(* IEC 61131-3 sources: F100R_S278_Temperville/MyController.device.xml.v3^/Plc Logic.plclogic.xml.v3^/Application.application.xml.v3^/03_Geral, 12 files *)

(* ---- B_Imagens.prg.st ---- *)
PROGRAM B_Imagens
VAR
	Index: INT;
END_VAR

//Imagens de Motores
ImgMotor[1]:=xMotorEntradaLigado;
ImgMotor[2]:=ImgMotor[2];
ImgMotor[3]:=xMotorFornoLigado;
ImgMotor[4]:=xMotorPassagemLigado;
ImgMotor[5]:=xMotorResfriadorLigado;
ImgMotor[6]:=xMotorSaidaLigado;
ImgMotor[7]:=xMotorDifusorSup01Ligado;
ImgMotor[8]:=xMotorDifusorInf01Ligado;
ImgMotor[9]:=xMotorDifusorSup02Ligado;
ImgMotor[10]:=xMotorDifusorInf02Ligado;
ImgMotor[11]:=xMotorGuilhotina01Ligado;
ImgMotor[12]:=xMotorGuilhotina02Ligado;
ImgMotor[13]:=xMotorLimpResfr02Ligado;
ImgMotor[14]:=xMotorCaixaFornoLigado;
ImgMotor[15]:=xMotorVentilador01Ligado;
ImgMotor[16]:=xMotorVentilador02Ligado;
ImgMotor[17]:=xMotorVentilador03Ligado;
ImgMotor[18]:=xMotorVentilador04Ligado;
ImgMotor[19]:=xMotorVentilador04Ligado;
ImgMotor[20]:=xMotorVentConvecEntLigado;
ImgMotor[21]:=xMotorVentConvecSaiLigado;
ImgMotor[22]:=xMotorGuilhotina01SupLigado;
ImgMotor[23]:=xMotorGuilhotina01InfLigado;
ImgMotor[24]:=xKaMotorOscilaResfr02Sup;
ImgMotor[25]:=xKaMotorOscilaResfr02Inf;

//Imagens de Válvula
ImgValvAberta[1]:=xSensorPortaEntrada;
ImgValvAberta[2]:=xSensorPortaSaida;
ImgValvAberta[3]:=xValvulaConveccaoLigada;
ImgValvAberta[4]:=xSensorGradeEntradaUp;
ImgValvAberta[5]:=xSensorGradeSaidaUp;

ImgValvFechada[1]:= NOT xSensorPortaEntrada;
ImgValvFechada[2]:= NOT xSensorPortaSaida;
ImgValvFechada[3]:= NOT xValvulaConveccaoLigada;
ImgValvFechada[4]:=	NOT xSensorGradeEntradaUp;
ImgValvFechada[5]:=	NOT xSensorGradeSaidaUp;

//Imagens Gerais
ImgGeral[1]:=xStatusNobreak;
ImgGeral[2]:=xBt01Emergencia; // Mesa Computador
ImgGeral[3]:=xBt02Emergencia; // Mesa Manual
ImgGeral[4]:=xBt03Emergencia; //
ImgGeral[5]:=xBt04Emergencia;
ImgGeral[6]:=xBt05Emergencia;
ImgGeral[7]:=xBt06Emergencia;
ImgGeral[8]:=xBt07Emergencia;
ImgGeral[9]:=xBt08Emergencia;
ImgGeral[10]:=xBt09Emergencia;
ImgGeral[11]:=xBt10Emergencia;
ImgGeral[12]:=xVentiladoresPainel;
ImgGeral[13]:=xVentiladoresSsr;
ImgGeral[14]:=xValvulaVeneziana;

FOR Index:=1 TO iNumResistencias DO
//	ImgRetornoSsrInferior[Index]:=xRetornoSsrInferior[Index];
//	ImgRetornoSsrSuperior[Index]:=xRetornoSsrSuperior[Index];
//	ImgResistenciaInferior[Index]:=xResistenciaInferior[Index];
//	ImgResistenciaSuperior[Index]:=xResistenciaSuperior[Index];
	ImgRetornoSsrInferior[Index]:=xResistenciaInferior[Index];
	ImgRetornoSsrSuperior[Index]:=xResistenciaSuperior[Index];
	ImgResistenciaHabilitadaInferior[Index]:=xResistenciaHabilitadaInferior[Index];
	ImgResistenciaHabilitadaSuperior[Index]:=xResistenciaHabilitadaSuperior[Index];
END_FOR

(* ---- C_Alarmes.prg.st ---- *)
PROGRAM C_Alarmes
VAR
	IndexAlm01: INT;
	AlmValvPortaEntrada: AlarmeValvula1vNeg;
	AlmValvPortaSaida: AlarmeValvula1vNeg;
	AlmGradeEntrada: AlarmeValvula1v;
	AlmGradeSaida: AlarmeValvula1v;
	TpAlmMotorSom: ARRAY[1..25] OF TP;
	TpAlmMotorSomIn: ARRAY[1..25] OF BOOL;
	TpAlmMotorSomQ: ARRAY[1..25] OF BOOL;
	AlmMotorSom: ARRAY[1..25] OF BOOL;
	AlarmeSom: TimerGeneration;
	AlarmeLum: TimerGeneration;
	xAlarmeSomEnable: BOOL;
	xAlarmeSomOut: BOOL;
	xAlarmeLumEnable: BOOL;
	xAlarmeLumOut: BOOL;
	TpRstSuper: TP;
	TpRstSuperiN: BOOL;
	TpRstSuperQ: BOOL;
	xAlarmeSonPortaEntradaForno: BOOL;
	xAlarmeSonPortaSaidaForno: BOOL;
	xAlarmeSonValvulaGradeEntrada: BOOL;
	xAlarmeSonValvulaGradeSaida: BOOL;
	xAlarmeGeralEncoder: BOOL;
	xAlarmeSonoroEncoderGeral: BOOL;
	xAlarmeGeralMotorParado: BOOL;
	xAlarmeSonoroMotorParadoGeral: BOOL;
	AlmMotoresBitsSoma: INT;
	AlmMotoresSonBitsSoma: INT;
END_VAR

AlmMotoresBitsSoma:=0;
AlmMotoresSonBitsSoma:=0;
FOR IndexAlm01:=1 TO 50 DO
	xAlarmesResistenciasGeralInferior[IndexAlm01]:=xAlarmeSsrInferiorFechado[IndexAlm01] OR xAlarmeSsrInferiorAberto[IndexAlm01] OR (*xAlarmeResistRompidaInferior[IndexAlm01]*) xFalhaForcadaInferior[IndexAlm01] OR xAlarmeResistForceInferior[IndexAlm01] OR AlmTermoparAbertoLogicoInf[IndexAlm01] OR AlmTemperaturaExcedeuLogicoInf[IndexAlm01];
	xAlarmesResistenciasGeralSuperior[IndexAlm01]:=xAlarmeSsrSuperiorFechado[IndexAlm01] OR xAlarmeSsrSuperiorAberto[IndexAlm01] OR (*xAlarmeResistRompidaSuperior[IndexAlm01]*) xFalhaForcadaSuperior[IndexAlm01] OR xAlarmeResistForceSuperior[IndexAlm01] OR AlmTermoparAbertoLogicoSup[IndexAlm01] OR AlmTemperaturaExcedeuLogicoSup[IndexAlm01];

	AlmMotoresBitsSoma:= AlmMotoresBitsSoma+ BOOL_TO_INT (AlmMotor[IndexAlm01]);

	TpAlmMotorSomIn[IndexAlm01]:=AlmMotor[IndexAlm01];
	TpAlmMotorSom[IndexAlm01](IN:=TpAlmMotorSomIn[IndexAlm01] , PT:=T#1S , Q=>TpAlmMotorSomQ[IndexAlm01] , ET=> );
	IF TpAlmMotorSomQ[IndexAlm01] THEN
		AlmMotorSom[IndexAlm01]:=TRUE;
	END_IF
	IF	bResetAlmGeral or xResetErro THEN
		AlmMotorSom[IndexAlm01]:=FALSE;
		AlmMotoresSonBitsSoma:=0;

	END_IF
	AlmMotoresSonBitsSoma:= AlmMotoresSonBitsSoma+ BOOL_TO_INT (AlmMotorSom[IndexAlm01]);

	xAlarmesTestesResistenciasInferiores[IndexAlm01]:=xTesteResistenciaInferiorFlh[IndexAlm01] OR xFalhaForcadaInferior[IndexAlm01] OR xAlarmeResistForceInferior[IndexAlm01];
	xAlarmesTestesResistenciasSuperiores[IndexAlm01]:=xTesteResistenciaSuperiorFlh[IndexAlm01] OR xFalhaForcadaSuperior[IndexAlm01] OR xAlarmeResistForceSuperior[IndexAlm01];

END_FOR;
xAlarmesMotores:= AlmMotoresBitsSoma>=1;
xAlarmesMotoresSon:= AlmMotoresSonBitsSoma>=1;

TpRstSuper(IN:=BtResetAlarmesGerais , PT:=T#500MS , Q=> TpRstSuperQ, ET=> );

bResetAlmGeral:=TpRstSuperQ OR xBtCalaAlarme ;
xBotaoResetaDrives:=TpRstSuperQ OR xBtCalaAlarme ;

IF BtResetAlarmesGerais THEN
	BtResetAlarmesGerais:=FALSE;
END_IF
//Alarmes de Motores

xAlarmeMotorEntrada	:=(xFalhaMotorEntrada OR xAlarmeCofInverMesaEntra);//AND NOT xPausaEmergenciaTof;
xAlarmeMotorForno	:=(xFalhaMotorForno OR xAlarmeCofInverMesaForno);//AND NOT xPausaEmergenciaTof;
xAlarmeMotorPass	:=(xFalhaMotorPassagem );//AND NOT xPausaEmergenciaTof;
xAlarmeMotorResfriador:=(xFalhaMotorResfriador OR xAlarmeCofInverMesaResfr);//AND NOT xPausaEmergenciaTof;
xAlarmeMotorSaida	:=(xFalhaMotorSaida OR xAlarmeCofInverMesaSaida);//AND NOT xPausaEmergenciaTof;
xAlarmeMotorDifusorInf01:=(xFalhaMotorDifusorInf01 );//AND NOT xPausaEmergenciaTof;
xAlarmeMotorDifusorSup01:=(xFalhaMotorDifusorSup01 );//AND NOT xPausaEmergenciaTof;
xAlarmeMotorDifusorInf02:=(xFalhaMotorDifusorInf02 );//AND NOT xPausaEmergenciaTof;
xAlarmeMotorDifusorSup02:=(xFalhaMotorDifusorSup02 OR xAlarmeCofInverResfrSup02);//AND NOT xPausaEmergenciaTof;
xAlarmeMotorGuilhotina01:=(xFalhaMotorGuilhotina01 );//AND NOT xPausaEmergenciaTof;
xAlarmeMotorGuilhotina02:=(xFalhaMotorGuilhotina02 OR xAlarmeCofInverGuilho02);//AND NOT xPausaEmergenciaTof;
xAlarmeMotorLimpResfr02:=(xFalhaMotorLimpResfr02 );//AND NOT xPausaEmergenciaTof;
xAlarmeMotorCaixaForno:=(xFalhaMotorCaixaForno OR xAlarmeCofInverCaixaForno);//AND NOT xPausaEmergenciaTof;
xAlarmeMotorVentilador01:=(xFalhaMotorVentilador01 );//AND NOT xPausaEmergenciaTof;
xAlarmeMotorVentilador02:=(xFalhaMotorVentilador02 );//AND NOT xPausaEmergenciaTof;
xAlarmeMotorVentilador03:=(xFalhaMotorVentilador03 OR xAlarmeCofInverVentila03);//AND NOT xPausaEmergenciaTof;
xAlarmeMotorVentilador04:=(xFalhaMotorVentilador04 );//AND NOT xPausaEmergenciaTof;
xAlarmeMotorVentConvecEnt:=(xFalhaMotorVentConvecEnt OR xAlarmeCofInverConvecEnt);//AND NOT xPausaEmergenciaTof;
xAlarmeMotorVentConvecSai:=(xFalhaMotorVentConvecSai );//AND NOT xPausaEmergenciaTof;
xAlarmeMotorGuilhotina01Sup:=(xFalhaMotorGuilhotina01Sup );//AND NOT xPausaEmergenciaTof;
xAlarmeMotorGuilhotina01Inf:=(xFalhaMotorGuilhotina01Inf );//AND NOT xPausaEmergenciaTof;

AlmMotor[1]:=xAlarmeMotorEntrada;
AlmMotor[2]:=AlmMotor[2];
AlmMotor[3]:=xAlarmeMotorForno;
AlmMotor[4]:=xAlarmeMotorPass;
AlmMotor[5]:=xAlarmeMotorResfriador;
AlmMotor[6]:=xAlarmeMotorSaida;
AlmMotor[7]:=xAlarmeMotorDifusorSup01;
AlmMotor[8]:=xAlarmeMotorDifusorInf01;
AlmMotor[9]:=xAlarmeMotorDifusorSup02;
AlmMotor[10]:=xAlarmeMotorDifusorInf02;
AlmMotor[11]:=xAlarmeMotorGuilhotina01;
AlmMotor[12]:=xAlarmeMotorGuilhotina02;
AlmMotor[13]:=AlmMotor[13];
AlmMotor[14]:=xAlarmeMotorCaixaForno;
AlmMotor[15]:=xAlarmeMotorVentilador01;
AlmMotor[16]:=xAlarmeMotorVentilador02;
AlmMotor[17]:=xAlarmeMotorVentilador03;
AlmMotor[18]:=xAlarmeMotorVentilador04;
AlmMotor[19]:=xAlarmeMotorBombaHidraulica;
AlmMotor[20]:=xAlarmeMotorVentConvecEnt;
AlmMotor[21]:=xAlarmeMotorVentConvecSai;
AlmMotor[22]:=xAlarmeMotorGuilhotina01Sup;
AlmMotor[23]:=xAlarmeMotorGuilhotina01Inf;
AlmMotor[24]:=xAlarmeMotorOscilaSup02;
AlmMotor[25]:=xAlarmeMotorOscilaInf02;

//Alarmes de Válvula

xSensorPortaEntradaAberta:=xSensorPortaEntrada;
xSensorPortaEntradaFechada:= NOT xSensorPortaEntrada;

AlmValvPortaEntrada(
	SensorValvAberta:= xSensorPortaEntradaAberta ,
	SensorValvFechad:= xSensorPortaEntradaFechada,
	AcionamentoValvula:= xValvPortaEntradaForno,// OR xOperacaoManual,
	ResetAlarm:=bResetAlmGeral OR xOperacaoManual,
	TempoAberto:= T#1500MS,
	TempoFechad:= T#1500MS,
	AlarmeValvAberta=> xAlarmePortaEntradaFornoAberta, //Porta não Abriu
	AlarmeValvFechada=> xAlarmePortaEntradaFornoFechada, // Porta não Fechou
	AlarmeSonoro=> xAlarmeSonPortaEntradaForno);

xAlarmePortaEntradaForno:=xAlarmePortaEntradaFornoAberta OR xAlarmePortaEntradaFornoFechada;

xSensorPortaSaidaAberta:=xSensorPortaSaida;
xSensorPortaSaidaFechada:= NOT xSensorPortaSaida;

AlmValvPortaSaida(
	SensorValvAberta:= xSensorPortaSaidaAberta ,
	SensorValvFechad:= xSensorPortaSaidaFechada,
	AcionamentoValvula:= xValvPortaSaidaForno,// OR xOperacaoManual,
	ResetAlarm:=bResetAlmGeral OR xOperacaoManual,
	TempoAberto:= T#2500MS,
	TempoFechad:= T#2000MS,
	AlarmeValvAberta=> xAlarmePortaSaidaFornoAberta, //Porta não Abriu
	AlarmeValvFechada=> xAlarmePortaSaidaFornoFechada, // Porta não Fechou
	AlarmeSonoro=> xAlarmeSonPortaSaidaForno);

xAlarmePortaSaidaForno:=xAlarmePortaSaidaFornoAberta OR xAlarmePortaSaidaFornoFechada;

// Alarme Grade Mesa de Entrada

xSensorGradeEntradaDown:= NOT xSensorGradeEntradaUp;

(*
AlmGradeEntrada(
	SensorValvAberta:= xSensorGradeEntradaUp,
	SensorValvFechad:= xSensorGradeEntradaDown,
	AcionamentoValvula:= xValvulaGradeEntrada,
	ResetAlarm:=bResetAlmGeral,
	TempoAberto:= T#2000MS,
	TempoFechad:= T#2000MS,
	AlarmeValvAberta=> xAlarmeValvulaGradeEntradaUp,
	AlarmeValvFechada=> xAlarmeValvulaGradeEntradaDown,
	AlarmeSonoro=>xAlarmeSonValvulaGradeEntrada);
*)
xAlarmeValvulaGradeEntrada:= xAlarmeValvulaGradeEntradaUp OR xAlarmeValvulaGradeEntradaDown;

// Alarme Grade Mesa de Saída

xSensorGradeSaidaDown:= NOT xSensorGradeSaidaUp;

AlmGradeSaida(
	SensorValvAberta:= xSensorGradeSaidaUp,
	SensorValvFechad:= xSensorGradeSaidaDown,
	AcionamentoValvula:= xValvulaGradeSaida,
	ResetAlarm:=bResetAlmGeral,
	TempoAberto:= T#5000MS,
	TempoFechad:= T#4000MS,
	AlarmeValvAberta=> xAlarmeValvulaGradeSaidaUp,
	AlarmeValvFechada=> xAlarmeValvulaGradeSaidaDown,
	AlarmeSonoro=> xAlarmeSonValvulaGradeSaida);

xAlarmeValvulaGradeSaida:= xAlarmeValvulaGradeSaidaUp OR xAlarmeValvulaGradeSaidaDown;

AlmValvAberta[1]:=xAlarmePortaEntradaFornoAberta;
AlmValvAberta[2]:=xAlarmePortaSaidaFornoAberta;
AlmValvAberta[3]:=xAlarmeValvulaGradeEntradaUp;
AlmValvAberta[4]:=xAlarmeValvulaGradeSaidaUp;
AlmValvAberta[5]:=AlmValvAberta[5];
AlmValvAberta[6]:=AlmValvAberta[6];
AlmValvAberta[7]:=AlmValvAberta[7];
AlmValvAberta[8]:=AlmValvAberta[8];
AlmValvAberta[9]:=AlmValvAberta[9];
AlmValvAberta[10]:=AlmValvAberta[10];

AlmValvFechada[1]:=xAlarmePortaEntradaFornoFechada;
AlmValvFechada[2]:=xAlarmePortaSaidaFornoFechada;
AlmValvFechada[3]:=xAlarmeValvulaGradeEntradaDown;
AlmValvFechada[4]:=xAlarmeValvulaGradeSaidaDown;
AlmValvFechada[5]:=AlmValvFechada[5];
AlmValvFechada[6]:=AlmValvFechada[6];
AlmValvFechada[7]:=AlmValvFechada[7];
AlmValvFechada[8]:=AlmValvFechada[8];
AlmValvFechada[9]:=AlmValvFechada[9];
AlmValvFechada[10]:=AlmValvFechada[10];

//Alarmes Gerais
AlmGeral[1]:=xAlarmePressaoArBaixaRede;
AlmGeral[2]:=xAlarmePressaoArAltaRede;
AlmGeral[3]:=xAlmNobreak;
AlmGeral[4]:=xSemEnergia;
AlmGeral[5]:=xLimpVidroForaPosicao;
AlmGeral[6]:=xAlmDisjGeral;
AlmGeral[7]:=xAlmDisjResist;
AlmGeral[8]:=xAlarmePressaoArBaixaMaq;
AlmGeral[9]:=xAlarmePressaoArAltaMaq;
AlmGeral[10]:=AlmGeral[10];

// Alarmes de Encoder
xAlarmeGeralEncoder:= xAlarmeGeralEncoderMeForno OR xAlarmeGeralEncoderMeResfriador (*OR xAlarmeGeralEncoderDuResfriadorSup01 OR xAlarmeGeralEncoderDuResfriadorInf01*) OR xAlarmeGeralEncoderDuResfriadorSup02 (*OR xAlarmeGeralEncoderDuResfriadorInf02 OR xAlarmeGeralEncoderGuiResfriador01*) OR xAlarmeGeralEncoderGuiResfriador02;
xAlarmeSonoroEncoderGeral:= xAlarmeSonoroEncoderMeForno OR xAlarmeSonoroEncoderMeResfriador (*OR xAlarmeSonoroEncoderDuResfriadorSup01 OR xAlarmeSonoroEncoderDuResfriadorInf01*) OR xAlarmeSonoroEncoderDuResfriadorSup02 (*OR xAlarmeSonoroEncoderDuResfriadorInf02 OR xAlarmeSonoroEncoderGuiResfriador01*) OR xAlarmeSonoroEncoderGuiResfriador02;

AlmEncoder[1]:=AlmEncoder[1];
AlmEncoder[2]:=xAlarmeGeralEncoderMeForno;
AlmEncoder[3]:=xAlarmeGeralEncoderMeResfriador;
AlmEncoder[4]:=xAlarmeGeralEncoderDuResfriadorSup01;
AlmEncoder[5]:=FALSE;//xAlarmeGeralEncoderDuResfriadorInf01;
AlmEncoder[6]:=xAlarmeGeralEncoderDuResfriadorSup02;
AlmEncoder[7]:=xAlarmeGeralEncoderDuResfriadorInf02;
AlmEncoder[8]:=xAlarmeGeralEncoderGuiResfriador01;
AlmEncoder[9]:=xAlarmeGeralEncoderGuiResfriador02;
AlmEncoder[10]:=FALSE;

// Alarmes Motor Parado por Falha Desconhecida

xAlarmeGeralMotorParado:=  xAlarmeMeFornoParado OR xAlarmeMeResfrParado;
xAlarmeSonoroMotorParadoGeral:= xAlarmeMeFornoParadoSom OR xAlarmeMeResfrParadoSom;

AlmMotorParado[1]:=AlmMotorParado[1];
AlmMotorParado[2]:=xAlarmeMeFornoParado;
AlmMotorParado[3]:=xAlarmeMeResfrParado;
AlmMotorParado[4]:=AlmMotorParado[4];
AlmMotorParado[5]:=AlmMotorParado[5];
AlmMotorParado[6]:=AlmMotorParado[6];
AlmMotorParado[7]:=AlmMotorParado[7];
AlmMotorParado[8]:=AlmMotorParado[8];
AlmMotorParado[9]:=AlmMotorParado[9];
AlmMotorParado[10]:=AlmMotorParado[10];

//Alerta Luminoso e Sonoro de Alarme

xAlarmeLumEnable:=xAlarmePortaEntradaForno OR xAlarmePortaSaidaForno OR xAlarmeValvulaGradeEntrada OR xAlarmeValvulaGradeSaida OR xAlarmesTermopares OR xAlarmesSSr OR xAlarmesMotores OR xAlarmePressaoArRede OR xAlarmePressaoArMaq OR xAlmNobreak OR xSemEnergia OR xAlmDisjGeral OR xAlmDisjResist OR xAlarmeGeralEncoder OR xAlarmeGeralMotorParado OR xLimpVidroForaPosicao OR xAlarmeSsrConvecEntSin OR xAlmTermoparAbertoConvecEntSin OR xAlmTemperExcedeuConvecEntSin;
AlarmeLum(ENABLE:=xAlarmeLumEnable , TIMELOW:=T#1S , TIMEHIGH:=T#1S , OUT=>xAlarmeLumOut );
//xAlarmeLuminoso:=xAlarmeLumOut OR xBtEmergencia OR NOT xReleSeguranca;
xSinalLumAmar:=xAlarmeLumOut;
xSinalLumVerm:=xBtEmergencia OR NOT xReleSeguranca OR xLedMotFornoStop;
xSinalLumVerd:= NOT xSinalLumVerm AND xLedMaqEmCiclo;

xAlarmeSomEnable:=xAlarmeSonPortaEntradaForno OR xAlarmeSonPortaSaidaForno OR xAlarmeSonValvulaGradeSaida OR xAlarmeSonValvulaGradeEntrada OR xAlarmesTermoparesSon OR xAlarmesSSrSon OR xAlarmesMotoresSon OR xAlarmePressaoArRedeSom OR xAlarmePressaoArMaqSom OR xAlmNobreakSom OR xAlmSomSemEnergia OR xAlmDisjGeralSom OR xAlmDisjResistSom OR xAlarmeSonoroEncoderGeral OR xAlarmeSonoroMotorParadoGeral OR xLimpVidroForaPosicaoSon OR xAlarmeSsrConvecEntSon OR xAlmTermoparAbertoConvecEntSon OR xAlmTemperExcedeuConvecEntSon;
AlarmeSom(ENABLE:=xAlarmeSomEnable , TIMELOW:=T#1S , TIMEHIGH:=T#1S , OUT=>xAlarmeSomOut );

xAlarmeSonoro:= (xAlarmeSomOut OR xSomDescarga OR xSomSemEnergia AND NOT xMotorCaixaFornoLigado) OR xAlertaSomCxForno;

(* ---- D_AnimaGeralResistencias.prg.st ---- *)
PROGRAM D_AnimaGeralResistencias
VAR
	Index: INT;
END_VAR

FOR Index:=1 TO iNumResistencias DO

//xAlarmesResistenciasGeral[Index]:=xAlarmeSsrInferiorFechado[Index] OR xAlarmeSsrInferiorAberto[Index] OR xAlarmeResistRompidaInferior[Index] OR AlmTermoparAbertoLogicoInf[Index] OR AlmTemperaturaExcedeuLogicoInf[Index];
//Inferior
	IF NOT xResistenciaHabilitadaInferior[Index] AND NOT xAlarmesResistenciasGeralInferior[Index] THEN
			iAnimaResistenciaInferior[Index]:=0;(*Resistência Desabilitada*)
	END_IF
	IF NOT xResistenciaInferior[Index] AND xResistenciaHabilitadaInferior[Index]THEN
			iAnimaResistenciaInferior[Index]:=1;(*Resistência Desligada*)
	END_IF
	IF xResistenciaInferior[Index] AND xResistenciaHabilitadaInferior[Index]THEN
			iAnimaResistenciaInferior[Index]:=2; (*Resistência Ligada*)
	END_IF
	IF xFalhaForcadaInferior[Index] OR  xAlarmesResistenciasGeralInferior[Index] (*xAlarmeResistForceSuperior[Index]*) THEN
			iAnimaResistenciaInferior[Index]:=3; (*Resistência Alarme*)
	END_IF

	IF AlmTermoparAbertoLogicoInf[Index] OR AlmTemperaturaExcedeuLogicoInf[Index] THEN
			iAnimaResistenciaInferior[Index]:=4; (*Termopar Alarme*)
	END_IF

	IF xResistenciaForcadaInferior[Index] AND ValorAmperagemResistenciaInferior[Index]>5 (*xResistenciaInferior[Index]*)  (*AND xResistenciaHabilitadaInferior[Index]*) THEN
			iAnimaResistenciaInferior[Index]:=5; (*Resistência Forçada*)
	END_IF

//Superior
	IF NOT xResistenciaHabilitadaSuperior[Index] AND NOT xAlarmesResistenciasGeralSuperior[Index] THEN
			iAnimaResistenciaSuperior[Index]:=0;(*Resistência Desabilitada*)
	END_IF
	IF NOT xResistenciaSuperior[Index] AND xResistenciaHabilitadaSuperior[Index]THEN
			iAnimaResistenciaSuperior[Index]:=1;(*Resistência Desligada*)
	END_IF
	IF (*(xReleSsrSuperior[Index] OR xSaidaReleRampaPatamarSup[Index])*)xResistenciaSuperior[Index] AND xResistenciaHabilitadaSuperior[Index]THEN
			iAnimaResistenciaSuperior[Index]:=2; (*Resistência Ligada*)
	END_IF
	IF xFalhaForcadaSuperior[Index] OR (*xAlarmeResistForceSuperior[Index]*) xAlarmesResistenciasGeralSuperior[Index] THEN
			iAnimaResistenciaSuperior[Index]:=3; (*Resistência Alarme*)
	END_IF
	IF AlmTermoparAbertoLogicoSup[Index] OR AlmTemperaturaExcedeuLogicoSup[Index] THEN
			iAnimaResistenciaSuperior[Index]:=4; (*Termopar Alarme*)
	END_IF
	IF xResistenciaForcadaSuperior[Index] AND ValorAmperagemResistenciaSuperior[Index]>5 (*xResistenciaSuperior[Index]*) (*AND xResistenciaHabilitadaSuperior[Index]*) THEN
			iAnimaResistenciaSuperior[Index]:=5; (*Resistência Forçada*)
	END_IF

END_FOR

(* ---- E_AnimaTesteGeralResistencias.prg.st ---- *)
PROGRAM E_AnimaTesteGeralResistencias
VAR
	Index: INT;
END_VAR

FOR Index:=1 TO iNumResistencias DO
//Inferior
	IF NOT xAlarmesResistenciasGeralInferior[Index] AND NOT xTesteResistenciaInferiorFlh[Index] AND NOT  xResistenciaInferior[Index] AND NOT xTestandoResistenciaInferior[Index]THEN
		iAnimaTesteResistenciaInferior[Index]:=0;(*Resistência Desligada*)
	END_IF

	IF xResistenciaForcadaInferior[Index] AND ValorAmperagemResistenciaInferior[Index]>40(*xResistenciaInferior[Index]*) THEN
		iAnimaTesteResistenciaInferior[Index]:=1; (*Resistência Forçada*)
	END_IF

	IF xResistenciaInferior[Index] AND xTestandoResistenciaInferior[Index]THEN
		iAnimaTesteResistenciaInferior[Index]:=2; (*Resistência Testando*)
	END_IF

	IF xTesteResistenciaInferiorOk[Index]THEN
		iAnimaTesteResistenciaInferior[Index]:=3; (* Teste Resistência Ok*)
	END_IF

	IF xFalhaForcadaInferior[Index] OR (*xAlarmeResistForceInferior[Index]*) xAlarmesResistenciasGeralInferior[Index] OR xTesteResistenciaInferiorFlh[Index] THEN
		iAnimaTesteResistenciaInferior[Index]:=4; (* Teste Resistência Resistência Alarme*)
	END_IF

//Superior
	IF NOT xAlarmesResistenciasGeralSuperior[Index] AND NOT xTesteResistenciaSuperiorFlh[Index] AND NOT xResistenciaSuperior[Index] AND NOT xTestandoResistenciaSuperior[Index]THEN
		iAnimaTesteResistenciaSuperior[Index]:=0;(*Resistência Desligada*)
	END_IF

	IF xResistenciaForcadaSuperior[Index] AND ValorAmperagemResistenciaSuperior[Index]>40(*xResistenciaSuperior[Index]*) THEN
		iAnimaTesteResistenciaSuperior[Index]:=1; (*Resistência Forçada*)
	END_IF

	IF xResistenciaSuperior[Index] AND xTestandoResistenciaSuperior[Index]THEN
		iAnimaTesteResistenciaSuperior[Index]:=2; (*Resistência Testando*)
	END_IF

	IF xTesteResistenciaSuperiorOk[Index]THEN
		iAnimaTesteResistenciaSuperior[Index]:=3; (* Teste Resistência Ok*)
	END_IF

	IF xFalhaForcadaSuperior[Index] OR (*xAlarmeResistForceSuperior[Index]*) xAlarmesResistenciasGeralSuperior[Index] OR xTesteResistenciaSuperiorFlh[Index] THEN
		iAnimaTesteResistenciaSuperior[Index]:=4; (* Teste Resistência Resistência Alarme*)
	END_IF

END_FOR

(* ---- F_AnimaAlmMotValv.prg.st ---- *)
PROGRAM F_AnimaAlmMotValv
VAR
	Index: INT;
END_VAR

FOR Index:=1 TO 25 DO
//Motores
	IF NOT AlmMotor[Index] AND NOT ImgMotor[Index] THEN
		iAnimaAlarmesMotores[Index]:=0; //Desligado
	END_IF
	IF NOT AlmMotor[Index] AND ImgMotor[Index] THEN
		iAnimaAlarmesMotores[Index]:=1; //Ligado
	END_IF
	IF AlmMotor[Index] THEN
		iAnimaAlarmesMotores[Index]:=2; //Alarme
	END_IF
//Válvulas

	IF (NOT AlmValvAberta[Index] OR NOT AlmValvFechada[Index] ) AND ImgValvFechada[Index] THEN
		iAnimaAlarmesValvulas[Index]:=0; // Fechada
	END_IF
	IF (NOT AlmValvAberta[Index] OR NOT AlmValvFechada[Index] ) AND ImgValvAberta[Index] THEN
		iAnimaAlarmesValvulas[Index]:=1; // Aberta
	END_IF
	IF AlmValvAberta[Index] OR AlmValvFechada[Index]  THEN
		iAnimaAlarmesValvulas[Index]:=2; // Alarme
	END_IF
END_FOR

(* ---- F_MensagemErroMotor.prg.st ---- *)
PROGRAM F_MensagemErroMotor
VAR
	Index: INT;
	sCodigoErroMotor: ARRAY[1..25] OF STRING;
	sDescricaoErroMotor: ARRAY[1..25] OF STRING;
END_VAR

FOR Index:=1 TO 20 DO
	IF wErroMotorId[Index]=4096 THEN
		sCodigoErroMotor[Index]:='OLF';
		sDescricaoErroMotor[Index]:='Sobrecarga Motor ';
	END_IF
	IF wErroMotorId[Index]=8976 THEN
		sCodigoErroMotor[Index]:='OCF';
		sDescricaoErroMotor[Index]:='Sobrecorrente Motor ';
	END_IF
	IF wErroMotorId[Index]=8992 THEN
		sCodigoErroMotor[Index]:='SCF';
		sDescricaoErroMotor[Index]:='Curto Circuito Motor ';
	END_IF
	IF wErroMotorId[Index]=9008 THEN
		sCodigoErroMotor[Index]:='SCF';
		sDescricaoErroMotor[Index]:='Curto Circuito Motor (Fase-Terra) ';
	END_IF
	IF wErroMotorId[Index]=9024 THEN
		sCodigoErroMotor[Index]:='SCF';
		sDescricaoErroMotor[Index]:='Curto Circuito Motor (Fase-Fase) ';
	END_IF
	IF wErroMotorId[Index]=12560 THEN
		sCodigoErroMotor[Index]:='OSF';
		sDescricaoErroMotor[Index]:='Sobretensão na Alimentação do Motor ';
	END_IF
	IF wErroMotorId[Index]=12576 THEN
		sCodigoErroMotor[Index]:='USF';
		sDescricaoErroMotor[Index]:='Sobretensão na Alimentação do Motor ';
	END_IF
	IF wErroMotorId[Index]=12592 THEN
		sCodigoErroMotor[Index]:='PHF';
		sDescricaoErroMotor[Index]:='Erro nas Fases de Alimentação ';
	END_IF
	IF wErroMotorId[Index]=13072 THEN
		sCodigoErroMotor[Index]:='OPF';
		sDescricaoErroMotor[Index]:='Erro nas Fases do Motor ';
	END_IF
	IF wErroMotorId[Index]=16912 THEN
		sCodigoErroMotor[Index]:='OHF';
		sDescricaoErroMotor[Index]:='Sobretemperatura no Motor ';
	END_IF
	IF wErroMotorId[Index]=21792 THEN
		sCodigoErroMotor[Index]:='EEF';
		sDescricaoErroMotor[Index]:='Erro na EEPROM ';
	END_IF
	IF wErroMotorId[Index]=24832 THEN
		sCodigoErroMotor[Index]:='InF';
		sDescricaoErroMotor[Index]:='Evento Interno ';
	END_IF
	IF wErroMotorId[Index]=33024 THEN
		sCodigoErroMotor[Index]:='COF';
		sDescricaoErroMotor[Index]:='Erro de Comunicação CANopen ';
	END_IF
	IF wErroMotorId[Index]=36864 THEN
		sCodigoErroMotor[Index]:='EPF';
		sDescricaoErroMotor[Index]:='Erro Externo ';
	END_IF

END_FOR

(* ---- F_SerialNumber.prg.st ---- *)
PROGRAM F_SerialNumber
VAR
	myCtr_Serial: DWORD;
	myCtr_Bateria: WORD;
	myCtr_ID: WORD;
	myCtr_FramesRx: UDINT;
	mCtr_Model: STRING(31);
END_VAR

//myCtr_Serial := M258.i_dwSerialNumber;
//myCtr_ID := M258.i_wVendorID;
//myCtr_FramesRx := SERIAL_R[0].i_udiFramesReceivedOK;

myCtr_Serial:=plc_r.i_dwSerialNumber;

myCtr_Bateria:=plc_r.i_wClockBatteryStatus;

mCtr_Model:=plc_r.i_sProductRef;

(* ---- O_VelocidadesMotores.prg.st ---- *)
PROGRAM O_VelocidadesMotores
VAR
	EntradaFornoGrosso: EquacaoDaReta;
	FornoResfriamentoGrosso: EquacaoDaReta;
	ResfriamentoSaidaGrosso: EquacaoDaReta;
	EntradaFornoFino: EquacaoDaReta;
	FornoResfriamentoFino: EquacaoDaReta;
	ResfriamentoSaidaFino: EquacaoDaReta;
	///Bloco Seleciona Pulsos para Vidro Fino ou Grosso
	SelecaoPulsos01: BlocoSelecaoEspessura;
	///Bloco Seleciona Pulsos para Vidro Fino ou Grosso
	SelecaoPulsos02: BlocoSelecaoEspessura;
	rVelocidadeMesaEntrada: REAL;
	rVelocidadeCargaMesaForno: REAL;
	rVelocidDescargaMesaForno: REAL;
	rVelocidCargaMesaResfriam: REAL;
	rVelocidDescargaMesaResfr: REAL;
	rVelocidadeMesaSaida: REAL;
	rVelocidadeMesaEntradaVidroFin: REAL;
	rVelocidadeCargaMesaFornoVidroFin: REAL;
	rVelocidDescargaMesaFornoVidroFin: REAL;
	rVelocidCargaMesaResfriamVidroFin: REAL;
	rVelocidDescargaMesaResfrVidroFin: REAL;
	rVelocidadeMesaSaidaVidroFin: REAL;
END_VAR

(* CÁLCULOS DOS VALORES DE VELOCIDADES DAS MESAS EM FUNÇÃO DA VELOCIDADE DO FORNO*)

//Vidros com Espessura 4mm
rVelocidadeCargaMesaFornoVidroFin:=INT_TO_REAL(iVelocidadeCargaFornoVidroFin);
rVelocidDescargaMesaFornoVidroFin:=INT_TO_REAL(iVelDescargaFornoVidroFin);
rVelocidDescargaMesaResfrVidroFin:=INT_TO_REAL(iVelDescargaResfriadorVidroFin);

EntradaFornoFino(
	rValorY:= (rVelocidadeCargaMesaFornoVidroFin/10),
	rPy1:= 25, //Velocidade y1 Inversor Forno
	rPy2:= 45, //Velocidade y2 Inversor Forno
	rPx1:= 39, //Velocidade x1 Inversor Entrada
	rPx2:= 70, //Velocidade x2 Inversor Entrada
	rValorX=> rVelocidadeMesaEntradaVidroFin);//Velocidade da Mesa de Entrada

iVelCargaMesaEntradaVidroFin:=REAL_TO_INT(rVelocidadeMesaEntradaVidroFin*10);
iVelCargaMeEntradaVidroFin:=iVelCargaMesaEntradaVidroFin+iCorretorCargaEntradaVidroFin;

FornoResfriamentoFino(
	rValorY:= (rVelocidDescargaMesaFornoVidroFin/10),
	rPy1:= 25,  //Velocidade y1 Inversor Forno
	rPy2:= 45,  //Velocidade y2 Inversor Forno
	rPx1:= 42.6, //Velocidade x1 Inversor Resfriador
	rPx2:= 77, //Velocidade x2 Inversor Resfriador
	rValorX=> rVelocidCargaMesaResfriamVidroFin);//Velocidade da Mesa do Resfriamento

iVelCargaResfriadorVidroFin:=REAL_TO_INT(rVelocidCargaMesaResfriamVidroFin*10);
iVelCargaMeResfriadorVidroFin:=iVelCargaResfriadorVidroFin+iCorretorCargaResfriadorVidroFin;

ResfriamentoSaidaFino(
	rValorY:= (rVelocidDescargaMesaResfrVidroFin/10),
	rPy1:= 42.6, // Velociade y1 Inversor Resfriador
	rPy2:= 77, // Velociade y2 Inversor Resfriador
	rPx1:= 37, // Velociade x1 Inversor Saída
	rPx2:= 65, // Velociade x2 Inversor Saída
	rValorX=> rVelocidadeMesaSaidaVidroFin); // Velocidade da Mesa de Saida

iVelCargaMesaSaidaVidroFin:=REAL_TO_INT(rVelocidadeMesaSaidaVidroFin*10);
iVelCargaMeSaidaVidroFin:=iVelCargaMesaSaidaVidroFin+iCorretorCargaSaidaVidroFin;

//-------------------------------------------------------------------------------//
//Vidros com Espessura Superior a 4mm
rVelocidadeCargaMesaForno:=INT_TO_REAL(iVelocidadeCargaForno);
rVelocidDescargaMesaForno:=INT_TO_REAL(iVelDescargaForno);
rVelocidDescargaMesaResfr:=INT_TO_REAL(iVelDescargaResfriador);

EntradaFornoGrosso(
	rValorY:= (rVelocidadeCargaMesaForno/10),
	rPy1:= 25, //Velocidade y1 Inversor Forno
	rPy2:= 40, //Velocidade y2 Inversor Forno
	rPx1:= 41.0, //Velocidade x1 Inversor Entrada
	rPx2:= 65.2, //Velocidade x2 Inversor Entrada
	rValorX=> rVelocidadeMesaEntrada);//Velocidade da Mesa de Entrada

iVelCargaMesaEntrada:=REAL_TO_INT(rVelocidadeMesaEntrada*10);
iVelCargaMeEntrada:=iVelCargaMesaEntrada+iCorretorCargaEntrada;

FornoResfriamentoGrosso(
	rValorY:= (rVelocidDescargaMesaForno/10),
	rPy1:= 25,  //Velocidade y1 Inversor Forno
	rPy2:= 40,  //Velocidade y2 Inversor Forno
	rPx1:= 46.2, //Velocidade x1 Inversor Resfriador
	rPx2:= 73.6, //Velocidade x2 Inversor Resfriador
	rValorX=> rVelocidCargaMesaResfriam);//Velocidade da Mesa do Resfriamento

iVelCargaResfriador:=REAL_TO_INT(rVelocidCargaMesaResfriam*10);
iVelCargaMeResfriador:=iVelCargaResfriador+iCorretorCargaResfriador;

ResfriamentoSaidaGrosso(
	rValorY:= (rVelocidDescargaMesaResfr/10),
	rPy1:= 46, // Velociade y1 Inversor Resfriador
	rPy2:= 73.6, // Velociade y2 Inversor Resfriador
	rPx1:= 45.5, // Velociade x1 Inversor Saída
	rPx2:= 72.2, // Velociade x2 Inversor Saída
	rValorX=> rVelocidadeMesaSaida); // Velocidade da Mesa de Saida

iVelCargaMesaSaida:=REAL_TO_INT(rVelocidadeMesaSaida*10);
iVelCargaMeSaida:=iVelCargaMesaSaida+iCorretorCargaSaida;

//Seleção das Variáveis de Velocidade

SelecaoPulsos01(
	xSelecao:= xEspessuraVidroFino,
	iEntrada0101:= iVelCargaMeEntradaVidroFin,
	iEntrada0102:= iVelCargaMeEntrada,
	iEntrada0201:= iVelocidadeCargaFornoVidroFin,
	iEntrada0202:= iVelocidadeCargaForno,
	iEntrada0301:= iVelVaiVemFornoVidroFin,
	iEntrada0302:= iVelVaiVemForno,
	iEntrada0401:= iVelDescargaFornoVidroFin,
	iEntrada0402:= iVelDescargaForno,
	iEntrada0501:= iVelCargaMeResfriadorVidroFin,
	iEntrada0502:= iVelCargaMeResfriador,
	iEntrada0601:= iVelVaiVemResfriadorVidroFin,
	iEntrada0602:= iVelVaiVemResfriador,
	iSaida01=> ,//iVelocidadeCargaMesaEntrada,
	iSaida02=> ,//iVelocidadeCargaMesaForno,
	iSaida03=> ,//iVelocidadeVaiVemMesaForno, Retirado para vir diretamente da Receita
	iSaida04=> ,//iVelocidadeDescargaMesaForno,
	iSaida05=> ,//iVelocidadeCargaMesaResfriador,
	iSaida06=> );//iVelocidadeVaiVemMesaResfriador);

SelecaoPulsos02(
	xSelecao:= xEspessuraVidroFino,
	iEntrada0101:= iVelDescargaResfriadorVidroFin,
	iEntrada0102:= iVelDescargaResfriador,
	iEntrada0201:= iVelCargaMeSaidaVidroFin,
	iEntrada0202:= iVelCargaMeSaida,
	iSaida01=> ,//iVelocidadeDescargaMesaResfriador,
	iSaida02=> );//iVelociadeCargaMesadeSaida);

(* ---- P_StatusOnline.prg.st ---- *)
PROGRAM P_StatusOnline

// STATUS PROCESSO

IF xFornoEmEspera THEN
	uStatusOperacao:=0; // Forno em Espera
END_IF
IF xFornoEmCiclo THEN
	uStatusOperacao:=1; // Forno em Ciclo
END_IF
IF xFornoFinalizando THEN
	uStatusOperacao:=2; // Forno Finalizando
END_IF

//STATUS MESA DE ENTRADA
uStatusMesaEntrada:=0; //Vazio

(*IF xCarregandoMesaEntrada THEN
	uStatusMesaEntrada:=1;
END_IF

IF xRetornaMesaEntrada THEN
	uStatusMesaEntrada:=2;
END_IF*)

//STATUS MESA DO FORNO

uStatusMesaForno:=0; //Vazio
IF xCarregandoForno THEN
	uStatusMesaForno:=1; //Carregando
END_IF
IF xFornoCarregado THEN
	uStatusMesaForno:=2; //Com Carga
END_IF
IF xDescarregandoForno THEN
	uStatusMesaForno:=3; //Descarregando
END_IF
IF xRetornandoForno THEN
	uStatusMesaForno:=4; //Retornando
END_IF

//STATUS MESA DO RESFRIAMENTO

uStatusMesaResfriador:=0; //Vazio
IF xCarregandoResfriador THEN
	uStatusMesaResfriador:=1; //Carregando
END_IF
IF xResfriadorCarregado THEN
	uStatusMesaResfriador:=2; //Com Carga
END_IF
IF xDescarregandoResfriador THEN
	uStatusMesaResfriador:=3; //Descarregando
END_IF

//STATUS MESA DE SAIDA

//STATUS DUCTOS INFERIOR 01
IF NOT xHomeDuctosResfriadorInf01Ok THEN
	uStatusDuctosResfriadorInf01:=0; // Efetuar Home
END_IF;

IF xDuctosInf01EmHome THEN
	uStatusDuctosResfriadorInf01:=1; // Em Home
END_IF

IF xDuctosInf01EmAjuste THEN
	uStatusDuctosResfriadorInf01:=2; // Ajustando Altura
END_IF

IF xAjusteAlturaDuctosInf01OK AND xHomeDuctosResfriadorInf01Ok THEN
	uStatusDuctosResfriadorInf01:=3; // Altura Ajustada
END_IF

IF xChAbreDuctosResfriadorInf01 THEN
	uStatusDuctosResfriadorInf01:=4; // Chave Acionada
END_IF;

IF xHomeDuctosResfriadorInf01Ok AND NOT xAjusteAlturaDuctosInf01OK AND NOT xDuctosInf01EmHome AND NOT xDuctosInf01EmAjuste AND NOT xChAbreDuctosResfriadorInf01 THEN
	uStatusDuctosResfriadorInf01:=5; // Ajustar Altura
END_IF;

//STATUS DUCTOS SUPERIOR 01
IF NOT xHomeDuctosResfriadorSup01Ok THEN
	uStatusDuctosResfriadorSup01:=0; // Efetuar Home
END_IF;

IF xDuctosSup01EmHome THEN
	uStatusDuctosResfriadorSup01:=1; // Em Home
END_IF

IF xDuctosSup01EmAjuste THEN
	uStatusDuctosResfriadorSup01:=2; // Ajustando Altura
END_IF

IF xAjusteAlturaDuctosSup01OK AND xHomeDuctosResfriadorSup01Ok THEN
	uStatusDuctosResfriadorSup01:=3; // Altura Ajustada
END_IF

IF xChAbreDuctosResfriadorSup01 THEN
	uStatusDuctosResfriadorSup01:=4; // Chave Acionada
END_IF;

IF xHomeDuctosResfriadorSup01Ok AND NOT xAjusteAlturaDuctosSup01OK AND NOT xDuctosSup01EmHome AND NOT xDuctosSup01EmAjuste AND NOT xChAbreDuctosResfriadorSup01 THEN
	uStatusDuctosResfriadorSup01:=5; // Ajustar Altura
END_IF;

//STATUS DUCTOS INFERIOR 02

IF NOT xHomeDuctosResfriadorInf02Ok THEN
	uStatusDuctosResfriadorInf02:=0; // Efetuar Home
END_IF;

IF xDuctosInf02EmHome THEN
	uStatusDuctosResfriadorInf02:=1; // Em Home
END_IF

IF xDuctosInf02EmAjuste THEN
	uStatusDuctosResfriadorInf02:=2; // Ajustando Altura
END_IF

IF xAjusteAlturaDuctosInf02OK AND xHomeDuctosResfriadorInf02Ok THEN
	uStatusDuctosResfriadorInf02:=3; // Altura Ajustada
END_IF

IF xChAbreDuctosResfriadorInf02 THEN
	uStatusDuctosResfriadorInf02:=4; // Chave Acionada
END_IF;

IF xHomeDuctosResfriadorInf02Ok AND NOT xAjusteAlturaDuctosInf02OK AND NOT xDuctosInf02EmHome AND NOT xDuctosInf02EmAjuste AND NOT xChAbreDuctosResfriadorInf02 THEN
	uStatusDuctosResfriadorInf02:=5; // Ajustar Altura
END_IF;

//STATUS DUCTOS SUPERIOR 02
IF NOT xHomeDuctosResfriadorSup02Ok THEN
	uStatusDuctosResfriadorSup02:=0; // Efetuar Home
END_IF;

IF xDuctosSup02EmHome THEN
	uStatusDuctosResfriadorSup02:=1; // Em Home
END_IF

IF xDuctosSup02EmAjuste THEN
	uStatusDuctosResfriadorSup02:=2; // Ajustando Altura
END_IF

IF xAjusteAlturaDuctosSup02OK AND xHomeDuctosResfriadorSup02Ok THEN
	uStatusDuctosResfriadorSup02:=3; // Altura Ajustada
END_IF

IF xChAbreDuctosResfriadorSup02 THEN
	uStatusDuctosResfriadorSup02:=4; // Chave Acionada
END_IF;

IF xHomeDuctosResfriadorSup02Ok AND NOT xAjusteAlturaDuctosSup02OK AND NOT xDuctosSup02EmHome AND NOT xDuctosSup02EmAjuste AND NOT xChAbreDuctosResfriadorSup02 THEN
	uStatusDuctosResfriadorSup02:=5; // Ajustar Altura
END_IF;

//STATUS GUILHOTINA 01

IF NOT xHomeGuilhotina01Ok THEN
	uStatusGuilhotina01:=0; // Efetuar Home
END_IF;

IF xGuilhotina01EmHome THEN
	uStatusGuilhotina01:=1; // Em Home
END_IF

IF xGuilhotina01EmAjuste THEN
	uStatusGuilhotina01:=2; // Ajustando Altura
END_IF

IF xAjusteAlturaGuilhotina01OK AND xHomeGuilhotina01Ok THEN
	uStatusGuilhotina01:=3; // Altura Ajustada
END_IF

IF xHomeGuilhotina01Ok AND NOT xAjusteAlturaGuilhotina01OK AND NOT xGuilhotina01EmHome AND NOT xGuilhotina01EmAjuste THEN
	uStatusGuilhotina01:=5; // Ajustar Altura
END_IF;

//STATUS GUILHOTINA 01 SUPERIOR

IF NOT xHomeGuilhotina01SupOk THEN
	uStatusGuilhotina01Sup:=0; // Efetuar Home
END_IF;

IF xGuilhotina01SupEmHome THEN
	uStatusGuilhotina01Sup:=1; // Em Home
END_IF

IF xGuilhotina01SupEmAjuste THEN
	uStatusGuilhotina01Sup:=2; // Ajustando Altura
END_IF

IF xAjusteAlturaGuilhotina01SupOK AND xHomeGuilhotina01SupOk THEN
	uStatusGuilhotina01Sup:=3; // Altura Ajustada
END_IF

IF xHomeGuilhotina01SupOk AND NOT xAjusteAlturaGuilhotina01SupOK AND NOT xGuilhotina01SupEmHome AND NOT xGuilhotina01SupEmAjuste THEN
	uStatusGuilhotina01Sup:=5; // Ajustar Altura
END_IF;

//STATUS GUILHOTINA 01 INFERIOR

IF NOT xHomeGuilhotina01InfOk THEN
	uStatusGuilhotina01Inf:=0; // Efetuar Home
END_IF;

IF xGuilhotina01InfEmHome THEN
	uStatusGuilhotina01Inf:=1; // Em Home
END_IF

IF xGuilhotina01InfEmAjuste THEN
	uStatusGuilhotina01Inf:=2; // Ajustando Altura
END_IF

IF xAjusteAlturaGuilhotina01InfOK AND xHomeGuilhotina01InfOk THEN
	uStatusGuilhotina01Inf:=3; // Altura Ajustada
END_IF

IF xHomeGuilhotina01InfOk AND NOT xAjusteAlturaGuilhotina01InfOK AND NOT xGuilhotina01InfEmHome AND NOT xGuilhotina01InfEmAjuste THEN
	uStatusGuilhotina01Inf:=5; // Ajustar Altura
END_IF;

//STATUS GUILHOTINA 02

IF NOT xHomeGuilhotina02Ok THEN
	uStatusGuilhotina02:=0; // Efetuar Home
END_IF;

IF xGuilhotina02EmHome THEN
	uStatusGuilhotina02:=1; // Em Home
END_IF

IF xGuilhotina02EmAjuste THEN
	uStatusGuilhotina02:=2; // Ajustando Altura
END_IF

IF xAjusteAlturaGuilhotina02OK AND xHomeGuilhotina02Ok THEN
	uStatusGuilhotina02:=3; // Altura Ajustada
END_IF

IF xHomeGuilhotina02Ok AND NOT xAjusteAlturaGuilhotina02OK AND NOT xGuilhotina02EmHome AND NOT xGuilhotina02EmAjuste THEN
	uStatusGuilhotina02:=5; // Ajustar Altura
END_IF;

(* ---- Q_MonitoraEncoder.prg.st ---- *)
PROGRAM Q_MonitoraEncoder
VAR
	MonitoraEncoderMForno: MonitoraEncoder;
	MonitoraEncoderMResfr: MonitoraEncoder;
	MonitoraEncoderResfrSup01: MonitoraEncoder;
	MonitoraEncoderGuilho01Sup: MonitoraEncoder;
	MonitoraEncoderGuilho01Inf: MonitoraEncoder;
	MonitoraEncoderResfrSup02: MonitoraEncoder;
	MonitoraEncoderGuilhotina02: MonitoraEncoder;
	xEncoderMesaFornoOk: BOOL;
	xEncoderMesaResfriamentoOk: BOOL;
	xEncoderResfriamentoSup01Ok: BOOL;
	xEncoderGuilhotina01SupOk: BOOL;
	xEncoderGuilhotina01InfOk: BOOL;
	xEncoderResfriamentoSup02Ok: BOOL;
	xEncoderGuilhotina02Ok: BOOL;
END_VAR

(* --------------- MONITORAMENTO DE ENCODERS ---------------- *)

MonitoraEncoderMForno(
	xEncoHabilitado:= xMotorFornoLigado AND NOT xAlarmeMotorForno AND NOT xAlarmeMeFornoParado AND NOT xTempoPausaRoletesOn,
	bResetAlmGeral:= bResetAlmGeral,
	tTempoCheck:=T#1000MS,
	dValorEncoder:= dValorEncoderFornoEntrada,
	xAlarmeEncoder=> xAlarmeGeralEncoderMeForno,
	xAlarmeSonoro=> xAlarmeSonoroEncoderMeForno,
	xEncoderOk=> 	xEncoderMesaFornoOk);

MonitoraEncoderMResfr(
	xEncoHabilitado:= xMotorResfriadorLigado,
	bResetAlmGeral:= bResetAlmGeral,
	tTempoCheck:=T#2000MS,
	dValorEncoder:= dValorEncoderResfrEntrada,
	xAlarmeEncoder=> xAlarmeGeralEncoderMeResfriador,
	xAlarmeSonoro=> xAlarmeSonoroEncoderMeResfriador,
	xEncoderOk=> xEncoderMesaResfriamentoOk);

MonitoraEncoderResfrSup02(
	xEncoHabilitado:= xMotorDifusorSup02Ligado,
	bResetAlmGeral:= bResetAlmGeral,
	tTempoCheck:=T#3000MS,
	dValorEncoder:= dValorEncoderDuctosResfriadorSup02,
	xAlarmeEncoder=> xAlarmeGeralEncoderDuResfriadorSup02,
	xAlarmeSonoro=> xAlarmeSonoroEncoderDuResfriadorSup02,
	xEncoderOk=> xEncoderResfriamentoSup02Ok);

MonitoraEncoderGuilhotina02(
	xEncoHabilitado:= xMotorGuilhotina02Ligado,
	bResetAlmGeral:= bResetAlmGeral,
	tTempoCheck:=T#1500MS,
	dValorEncoder:= dValorEncoderGuilhotinaResfriador02,
	xAlarmeEncoder=> xAlarmeGeralEncoderGuiResfriador02,
	xAlarmeSonoro=>xAlarmeSonoroEncoderGuiResfriador02,
	xEncoderOk=>xEncoderGuilhotina02Ok);

(* ---- R_MonitoraMotores.prg.st ---- *)
PROGRAM R_MonitoraMotores
VAR
	AlarmeMotorMeFornoStop: AlarmeMotorParado;
	AlarmeMotorMeResfrStop: AlarmeMotorParado;
	AlarmeMotorFornoParadoEncoder: MonitoraEncoder;
	PulsoLedMotFornoStop: TimerGeneration;
	xMotorMeFornoStop: BOOL;
	xMotorMeResfrStop: BOOL;
	xAlarmeMeFornoParadoEncoder: BOOL;
	xAlarmeParadoMotorMesaForno: BOOL;
END_VAR

AlarmeMotorFornoParadoEncoder(
	xEncoHabilitado:= xFornoEmCicloComCarga AND NOT xTempoPausaRoletesOn,
	bResetAlmGeral:= bResetAlmGeral,
	tTempoCheck:=T#1000MS,
	dValorEncoder:= dValorEncoderFornoEntrada,
	xAlarmeEncoder=> xAlarmeMeFornoParadoEncoder,
	xAlarmeSonoro=> ,
	xEncoderOk=> 	);

xAlarmeParadoMotorMesaForno:= NOT xMotorFornoLigado AND NOT xOperacaoManual AND NOT xTempoPausaRoletesOn AND NOT xDesligaMotorFornoTempBaixa AND xEnergiaOk AND NOT xPause;
xMotorMeFornoStop:= xAlarmeParadoMotorMesaForno OR xAlarmeMeFornoParadoEncoder;
AlarmeMotorMeFornoStop(KaMotor:=xMotorMeFornoStop , ResetAlarm:=bResetAlmGeral , AlarmeMotor=> xAlarmeMeFornoParado, AlarmeSonoro=>xAlarmeMeFornoParadoSom );

PulsoLedMotFornoStop(ENABLE:= xMotorMeFornoStop, TIMELOW:=T#500MS , TIMEHIGH:=T#500MS , OUT=>xLedMotFornoStop );

xMotorMeResfrStop:= xMesaResfriadorOn AND NOT xMotorResfriadorLigado AND NOT xOperacaoManual AND xEnergiaOk AND NOT xPausaEmergencia  AND NOT xPausaResfrChAbreSupAcionanda;
AlarmeMotorMeResfrStop(KaMotor:=xMotorMeResfrStop , ResetAlarm:=bResetAlmGeral , AlarmeMotor=> xAlarmeMeResfrParado, AlarmeSonoro=>xAlarmeMeResfrParadoSom );

(* ---- S_Termocamera.prg.st ---- *)
PROGRAM S_Termocamera
VAR
	MediaValoresTermocam: RegistradorMedia;
	rValorTemperTermocamera: REAL;
	rTemperaturaTermocameralocal: REAL;
END_VAR

MediaValoresTermocam.rDadoEntrada:=INT_TO_REAL(iValorTemperTermocamera);

MediaValoresTermocam(rDadoEntrada:= , rDadoSaida=>rValorTemperTermocamera );

rTemperaturaTermocamera:= (32767/rValorTemperTermocamera);

rTemperaturaTermocameralocal:=(rValorTemperTermocamera/32767);
